(* IEC 61131-3 sources: actuators/src/Endswitch, 6 files *)

(* ---- EndswitchBehavior.st ---- *)
USING Simatic.Ax.Commands;

NAMESPACE Simatic.Ax.Actuators

    // Enumeration representing the behavior of an endswitch.
    TYPE
        EndswitchBehavior : (NormallyOpen, NormallyClosed) := NormallyOpen;
    END_TYPE

END_NAMESPACE

(* ---- SuperVisionMode.st ---- *)
NAMESPACE Simatic.Ax.Actuators
    TYPE
        SuperVisionMode : (None, PositionControl, Action, Reaction) := None;
    END_TYPE

    TYPE
        /// Represents different types of supervision errors that can occur in the system.
        /// None: No error has occurred.
        /// PositionError: Indicates an unexpected change in the actuator's position.
        /// ActionError: Indicates that no action occurred after initiating a command, such as MoveToWorkPosition, and the current position was not left.
        /// ReactionError: Indicates that the target position was not reached, despite the command being executed.
        SuperVisionError : WORD (None := WORD#16#0000, Evaluating := WORD#16#7001, PositionError := WORD#16#8001, ActionError := WORD#16#8002, ReactionError := WORD#16#8003) := None;
    END_TYPE
END_NAMESPACE

(* ---- itfBooleanUpdate.st ---- *)
USING System.Timer;
USING Simatic.Ax.IO.Input;
NAMESPACE Simatic.Ax.Actuators

    INTERFACE itfBooleanUpdate
        // Reads the cyclic signal and updates the internal state of the endswitch.
        METHOD Update
            VAR_INPUT
                signal : BOOL;       // Current signal state.
                valid : BOOL := TRUE; // Indicates if the signal is valid.
                default : BOOL := FALSE; // Default signal state.
            END_VAR
        END_METHOD
    END_INTERFACE

END_NAMESPACE

(* ---- itfEndswitch.st ---- *)
USING System.Timer;

NAMESPACE Simatic.Ax.Actuators

    // Interface for an endswitch, defining methods for monitoring and retrieving its state.
    INTERFACE itfEndswitch
        // Starts monitoring the endswitch with a specified monitoring time.
        METHOD StartMonitoring
            VAR_INPUT
                MonitoringTime : LTIME; // Duration for monitoring.
            END_VAR
        END_METHOD

        // Checks if the endswitch is currently activated.
        METHOD IsActivated : BOOL
        END_METHOD

        // Checks if the endswitch has been reached.
        METHOD HasReached : BOOL
        END_METHOD

        // Checks if the endswitch has been left.
        METHOD HasLeft : BOOL
        END_METHOD

        // Checks if the monitoring time has elapsed.
        METHOD TimeHasElapsed : BOOL
        END_METHOD
    END_INTERFACE
END_NAMESPACE

(* ---- Endswitch.st ---- *)
USING NotificationService.ErrorHandling;
USING System.Timer;
USING Simatic.Ax.IO.Input;
USING NotificationService.ErrorHandling;
NAMESPACE Simatic.Ax.Actuators
    /// Class representing an endswitch, implementing the itfEndswitch interface.
    /// Input: None.
    /// Returns: Provides supervision and monitoring capabilities for an endswitch.
    CLASS BooleanEndswitch EXTENDS ErrorProviderBase IMPLEMENTS itfEndswitch, itfBooleanUpdate
        VAR PUBLIC
            /// Defines whether the endswitch is normally open or closed.
            Behavior : EndswitchBehavior;

            /// Supervision time for action errors.
            SuperVisionTimeAction : LTIME := T#1s;

            /// Supervision time for reaction errors.
            SuperVisionTimeReaction : LTIME := T#5s;
        END_VAR

        VAR
            /// Binary signal for the endswitch.
            _binSignal : BinSignal;

            /// Timer for monitoring the endswitch.
            _monTimer : Ondelay;

            /// Current error state of the endswitch.
            _errorState : SuperVisionState;

            /// Current supervision mode of the endswitch.
            _superVisionMode : SuperVisionMode;

            /// Indicates if the endswitch is initialized.
            _isInitialized : BOOL;

            /// Indicates if the endswitch has been left.
            _hasLeft : BOOL;

            /// Indicates if the endswitch has been reached.
            _hasReached : BOOL;
            _isActivated : BOOL;
            /// Alarm object for reporting errors.
            _Alarm : Alarm := (id := '4711', errorMessage := 'Endswitch fault');

            /// Counter for the number of errors detected.
            _errorCount : DINT;
            _hasLeftCounter : DINT;
            _hasReachedCounter : DINT;
        END_VAR

        /// Reads the cyclic signal and updates the internal state of the endswitch.
        /// Input: signal - Current signal state.
        ///        valid - Indicates if the signal is valid.
        ///        default - Default signal state.
        /// Returns: None.
        METHOD PUBLIC Update
            VAR_INPUT
                /// Current signal state.
                signal : BOOL;

                /// Indicates if the signal is valid.
                valid : BOOL := TRUE;

                /// Default signal state.
                default : BOOL := FALSE;
            END_VAR

            _binSignal.invert := Behavior = EndswitchBehavior#NormallyClosed;
            _binSignal.ReadCyclic(signal := signal, valid := valid, default := default);
            _isActivated := _binSignal.Q();
            _hasLeft := _binSignal.QFal();
            _hasReached := _binSignal.QRis();
            _monTimer();
            _errorState := THIS.Check();
        END_METHOD

        /// Evaluates the current state of the endswitch and determines if a supervision error has occurred.
        /// Supervision errors include:
        /// - None: No error has occurred.
        /// - PositionError: The actuator's position changed unexpectedly.
        /// - ActionError: No action occurred after initiating a command, and the current position was not left.
        /// - ReactionError: The target position was not reached despite the command being executed.
        METHOD PRIVATE Check : SuperVisionState
            CASE _superVisionMode OF
                SuperVisionMode#None:
                    _monTimer(signal := FALSE);
                    Check := _errorState;
                SuperVisionMode#Reaction:
                    Check := SuperVisionState#EvaluatingRecaction;
                    IF (_hasReached) THEN
                        _hasReachedCounter := _hasReachedCounter + 1;
                        _superVisionMode := SuperVisionMode#None;
                    END_IF;
                    // Error
                    IF _monTimer.output THEN
                        _Alarm.errorMessage := 'Target position not reached (Reaction Error)';
                        THIS.Notify(e := _Alarm);
                        _errorCount := _errorCount + 1;
                        Check := SuperVisionState#ReactionError;
                        _superVisionMode := SuperVisionMode#None;
                    END_IF;
                SuperVisionMode#Action:
                    Check := SuperVisionState#EvaluatingAction;
                    IF (_hasLeft) THEN
                        _hasLeftCounter := _hasLeftCounter + 1;
                        _superVisionMode := SuperVisionMode#None;
                    END_IF;
                    // Error
                    IF _monTimer.output THEN
                        _Alarm.errorMessage := 'No action occurred after command initiation (Action Error)';
                        THIS.Notify(e := _Alarm);
                        _errorCount := _errorCount + 1;
                        _monTimer(signal := FALSE);
                        Check := SuperVisionState#ActionError;
                        _superVisionMode := SuperVisionMode#None;
                    END_IF;
                SuperVisionMode#PositionControl:
                    Check := SuperVisionState#EvaluatingPosition;
                    IF _hasReached OR _hasLeft THEN
                        _Alarm.errorMessage := 'Unexpected position change detected (Position Error)';
                        THIS.Notify(e := _Alarm);
                        _errorCount := _errorCount + 1;
                        _superVisionMode := SuperVisionMode#None;
                        Check := SuperVisionState#PositionError;
                    END_IF;
            END_CASE;
            ;
        END_METHOD

        /// Returns the error status of the endswitch.
        /// Input: None.
        /// Returns: The current supervision error state of the endswitch.
        METHOD PUBLIC GetError : SuperVisionState
            GetError := _errorState;
        END_METHOD

        /// Starts monitoring the endswitch with a specified monitoring time.
        METHOD PUBLIC EnableSupervision
            VAR_INPUT
                /// The supervision mode to enable.
                Mode : SuperVisionMode;
            END_VAR
            _errorState := SuperVisionState#None;
            _superVisionMode := Mode;
            _monTimer(signal := FALSE);
            CASE _superVisionMode OF
                SuperVisionMode#Reaction:
                    _monTimer(signal := TRUE, duration := SuperVisionTimeReaction);
                SuperVisionMode#Action:
                    _monTimer(signal := TRUE, duration := SuperVisionTimeAction);
                SuperVisionMode#PositionControl:
                    ;
                ELSE;
                    ;
            END_CASE;
        END_METHOD

        /// Checks if the monitoring time has elapsed.
        METHOD PUBLIC TimeHasElapsed : BOOL
            TimeHasElapsed := _monTimer.output;
        END_METHOD

        /// Checks if the endswitch is currently activated.
        METHOD PUBLIC IsActivated : BOOL
            IsActivated := _binSignal.Q();
            ;
        END_METHOD

        /// Checks if the endswitch has been reached.
        METHOD PUBLIC HasReached : BOOL
            HasReached := _binSignal.QRis();
            ;
        END_METHOD

        /// Checks if the endswitch has been left.
        METHOD PUBLIC HasLeft : BOOL
            HasLeft := _binSignal.QFal();
            ;
        END_METHOD
    END_CLASS

END_NAMESPACE

(* ---- NullEndswitch.st ---- *)
USING System.Timer;

NAMESPACE Simatic.Ax.Actuators

    // Dummy implementation of the ItfEndswitch interface for testing purposes.
    CLASS INTERNAL NullEndswitch IMPLEMENTS itfEndswitch
        VAR PUBLIC
            MonitoringTime : LTIME := T#5s; // Default monitoring time.
        END_VAR

        VAR
            _monTimer : Ondelay;       // Timer for monitoring.
            _hasActivated : BOOL;     // Indicates if the endswitch has been activated.
            _hasLeft : BOOL;          // Indicates if the endswitch has been left.
            _activatedOld : BOOL;     // Previous activation state.
        END_VAR

        // Reads the cyclic signal and updates the internal state of the dummy endswitch.
        METHOD PUBLIC ReadCyclic
            _monTimer();
            _hasActivated := _monTimer.output AND NOT(_activatedOld);
            _hasLeft := NOT(_monTimer.output) AND _activatedOld;
            _activatedOld := _monTimer.output;
        END_METHOD

        // Starts monitoring the dummy endswitch with a specified monitoring time.
        METHOD PUBLIC StartMonitoring
            VAR_INPUT
                MonitoringTime : LTIME := T#5S; // Default monitoring time.
            END_VAR

            _monTimer(signal := FALSE);
            _monTimer(signal := TRUE, duration := MonitoringTime);
            ;
        END_METHOD

        // Checks if the monitoring time has elapsed.
        METHOD PUBLIC TimeHasElapsed : BOOL
            TimeHasElapsed := FALSE;
        END_METHOD

        // Checks if the dummy endswitch is currently activated.
        METHOD PUBLIC IsActivated : BOOL
            IsActivated := _monTimer.output;
        END_METHOD

        // Checks if the dummy endswitch has been reached.
        METHOD PUBLIC HasReached : BOOL
            HasReached := _hasActivated;
        END_METHOD

        // Checks if the dummy endswitch has been left.
        METHOD PUBLIC HasLeft : BOOL
            HasLeft := _hasLeft;
            ;
        END_METHOD
    END_CLASS
END_NAMESPACE
